{attribute 'GeneratedUsingTerminal: EL2522-0000-0017'}
{attribute addProperty BoxType "EL2522-0000-0017"}
{attribute addProperty Id "Target_counter_valueAT %Q*UDINT4"}
{attribute addProperty CRC "527260614"}
{attribute addProperty Size "4"}
TYPE PTO_Target_Channel_1F6D5BC6 :
STRUCT
	{attribute addProperty Name "Target_counter_value"}
	Target_counter_value AT %Q* : UDINT;
END_STRUCT
END_TYPE

(* stored: Version 1.2.0.0, ProductVersion 3.1.4024.9
   DUT PTO_Target_Channel_1F6D5BC6: Id {07f42afe-8bf9-4fd1-b0bd-20c6cdbd5a22} *)
